DATA_BLOCK "dbArchiveEquipDoor"
{ S7_Optimized_Access := 'TRUE' }
VERSION : 0.8
NON_RETAIN
"fbArchiveEquipDoor"

BEGIN

END_DATA_BLOCK

